FUNCTION_BLOCK Motor_FB
VAR
END_VAR

METHOD M_Delay : BOOL
VAR_INPUT
END_VAR
END_METHOD

METHOD PUBLIC M_Start : BOOL
VAR_INPUT
END_VAR
END_METHOD

METHOD M_Stop : BOOL
VAR_INPUT
END_VAR
END_METHOD

END_FUNCTION_BLOCK

(* stored: Version 1.1.0.1, ProductVersion 3.1.4024.12
   POU Motor_FB: Id {9b3ada02-ffd2-4e0a-9396-9cd5f8ad298b}, SpecialFunc None
   Method M_Delay: Id {eb52c425-d85a-487e-94c7-f839f48eecf7}
   Method M_Start: Id {d1c8712d-a0e9-45aa-915c-8b3841d464bd}
   Method M_Stop: Id {3e665fa6-4a1d-4c20-82c6-daca24e7ff33} *)
